RoboDK station: IndustrialRobot.rdk

Station IndustrialRobot (saved by RoboDK 6.0.1). Poses are relative to the parent item; angles as X-Y-Z fixed-axis rotations.
